FUNCTION_BLOCK Cylinder
VAR_INPUT
	bExecute: BOOL;
	command_activate: BOOL;
	push_edge_time: TIME := T#0.5S;
	pull_edge_time: TIME := T#0.5S;
	limit_time	: TIME := T#3S;
	keep_actuator : BOOL := FALSE;
	stroke_wait_time: TIME := T#5S;
END_VAR
VAR_OUTPUT
	status: position_status := position_status.unknown;
	position: _2_position;
	current_position: UINT;
	bError:BOOL;
END_VAR
VAR
	push_command: BOOL;
	pull_command: BOOL;
	edge_timer:Tc2_Standard.TON;
	limit_timer:Tc2_Standard.TON;
	stroke_wait_timer: Tc2_Standard.TON;
	last_cycle_position: _2_position;
	last_cycle_status : position_status;
END_VAR

VAR_IN_OUT
	io: cylinder2IO;
END_VAR

IF bExecute THEN
	stroke_wait_timer(IN := last_cycle_position = position, PT := stroke_wait_time);
	CASE position OF
		_2_position.position_2:
			IF stroke_wait_timer.Q THEN
				push_command := FALSE;
				pull_command := TRUE;				
			END_IF
		_2_position.position_1:
			IF stroke_wait_timer.Q THEN
				push_command := TRUE;
				pull_command := FALSE;
			END_IF
	END_CASE
ELSE
	push_command := FALSE;
	pull_command := FALSE;
END_IF
last_cycle_position := position;

command_activate := push_command OR pull_command;
CASE status OF
	position_status.unknown:
		IF last_cycle_status = position_status.inposition THEN
			bError := TRUE;
		END_IF
		io.push_output := FALSE;
		io.pull_output := FALSE;
		IF bError THEN
			bError := command_activate;
		ELSE
			IF push_command AND position = _2_position.position_1 THEN
				status := position_status.moving;
			END_IF
			IF pull_command AND position = _2_position.position_2 THEN
				status := position_status.moving;
			END_IF
		END_IF
	position_status.inposition:
		edge_timer.IN := FALSE;
		
		CASE position OF
			_2_position.position_1:
				IF push_command	THEN
					status := position_status.moving;
				END_IF
				IF io.push_sensor OR NOT io.pull_sensor THEN
					status := position_status.unknown;
				END_IF
			_2_position.position_2:
				IF pull_command	THEN
					status := position_status.moving;
				END_IF
				IF NOT io.push_sensor OR io.pull_sensor THEN
					status := position_status.unknown;
				END_IF
		END_CASE
		
		IF keep_actuator THEN
			io.push_output := (position = _2_position.position_2);
			io.pull_output := (position = _2_position.position_1);
		ELSE
			io.push_output := FALSE;
			io.pull_output := FALSE;
		END_IF
		
	position_status.moving:
		IF push_command THEN
			edge_timer.PT := push_edge_time;
			IF io.push_sensor AND NOT io.pull_sensor THEN
				edge_timer.IN := TRUE;
				IF edge_timer.Q THEN
					position := _2_position.position_2;
					status := position_status.inposition;
				END_IF
			ELSE
				edge_timer.IN := FALSE;
			END_IF
			io.push_output := TRUE;
			io.pull_output := FALSE;
		END_IF
		IF pull_command THEN
			edge_timer.PT := pull_edge_time;
			IF NOT io.push_sensor AND io.pull_sensor THEN
				edge_timer.IN := TRUE;
				IF edge_timer.Q THEN
					position := _2_position.position_1;
					status := position_status.inposition;
				END_IF
			ELSE
				edge_timer.IN := FALSE;
			END_IF
			io.push_output := FALSE;
			io.pull_output := TRUE;
		END_IF

END_CASE


limit_timer(IN:=command_activate AND (status <> position_status.inposition), PT:=limit_time);
IF limit_timer.Q THEN
	status := position_status.unknown;
	bError := TRUE;
END_IF

edge_timer();

last_cycle_status := status;

END_FUNCTION_BLOCK

(* stored: Version 1.1.0.1, ProductVersion 3.1.4024.12
   POU Cylinder: Id {78da19cc-508f-4a31-91e7-b419e493c65e}, SpecialFunc None *)
